Omron CX-Programmer project NewProject (CX-Programmer 9.75)

# PLC NewPLC1: CJ1M CPU21
I/O table (CPU CJ1M-CPU21): rack 0 slot 0 CJ1W-OC211; rack 0 slot 1 CJ1W-ID211; rack 0 slot 2 CJ1W-AD041-V1

## Global symbols (name address type ; comment)
100.00 BOOL  ; SET tajmer za miksovanje
200.00 BOOL  ; Ukljucuje se
T0001 BOOL  ; Tajmer potreban da se smesa miksuje
T0002 BOOL  ; Tajmer potreban da se isprazni rezervoar

## Program NewProgram1 (cyclic task 0)
Local symbols
M_1 2961.04 BOOL  ; Mikser
ON_OFF 2960.04 BOOL  ; ON/OFF prekidac
S_1 2960.00 BOOL  ; Ultrazvucni senzor
S_2 2960.01 BOOL  ; Senzor za nivo vode
S_3 2960.02 BOOL  ; Senzor za nivo cementa
S_4 2960.03 BOOL  ; Senzor za nivo peska
V_1 2961.00 BOOL  ; Ventil za vodu
V_2 2961.01 BOOL  ; Ventil za cement
V_3 2961.02 BOOL  ; Ventil za pesak
V_4 2961.03 BOOL  ; Ventil za ispustanje smese

### Section Section1

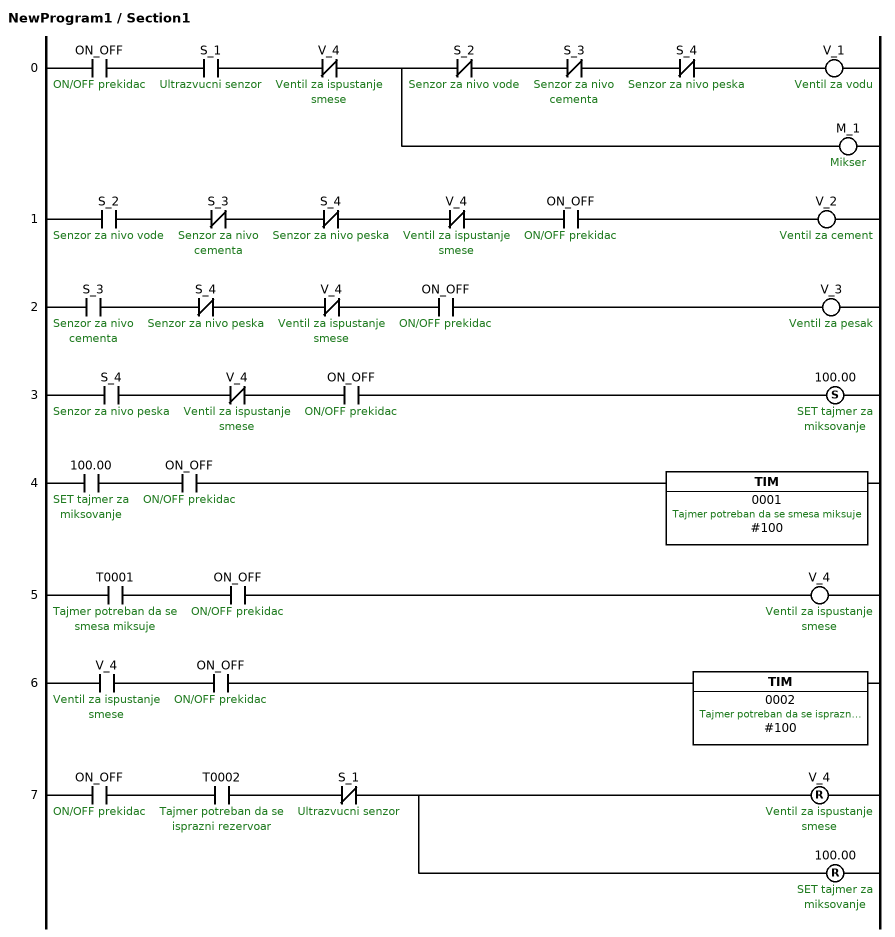
; rung 0
LD ON_OFF  ; ON/OFF prekidac
AND S_1  ; Ultrazvucni senzor
ANDNOT V_4  ; Ventil za ispustanje smese
OUT TR0
ANDNOT S_2  ; Senzor za nivo vode
ANDNOT S_3  ; Senzor za nivo cementa
ANDNOT S_4  ; Senzor za nivo peska
OUT V_1  ; Ventil za vodu
LD TR0
OUT M_1  ; Mikser
; rung 1
LD S_2  ; Senzor za nivo vode
ANDNOT S_3  ; Senzor za nivo cementa
ANDNOT S_4  ; Senzor za nivo peska
ANDNOT V_4  ; Ventil za ispustanje smese
AND ON_OFF  ; ON/OFF prekidac
OUT V_2  ; Ventil za cement
; rung 2
LD S_3  ; Senzor za nivo cementa
ANDNOT S_4  ; Senzor za nivo peska
ANDNOT V_4  ; Ventil za ispustanje smese
AND ON_OFF  ; ON/OFF prekidac
OUT V_3  ; Ventil za pesak
; rung 3
LD S_4  ; Senzor za nivo peska
ANDNOT V_4  ; Ventil za ispustanje smese
AND ON_OFF  ; ON/OFF prekidac
SET 100.00  ; SET tajmer za miksovanje
; rung 4
LD 100.00  ; SET tajmer za miksovanje
AND ON_OFF  ; ON/OFF prekidac
TIM 0001 #100  ; Tajmer potreban da se smesa miksuje
; rung 5
LD T0001  ; Tajmer potreban da se smesa miksuje
AND ON_OFF  ; ON/OFF prekidac
OUT V_4  ; Ventil za ispustanje smese
; rung 6
LD V_4  ; Ventil za ispustanje smese
AND ON_OFF  ; ON/OFF prekidac
TIM 0002 #100  ; Tajmer potreban da se isprazni rezervoar
; rung 7
LD ON_OFF  ; ON/OFF prekidac
AND T0002  ; Tajmer potreban da se isprazni rezervoar
ANDNOT S_1  ; Ultrazvucni senzor
RSET V_4  ; Ventil za ispustanje smese
RSET 100.00  ; SET tajmer za miksovanje

### Section END
; rung 0
END(001)